FUNCTION_BLOCK AR_CLIENT_1_0 (* Send a REAL from an AR adapter as a remote OPC-UA write via CLIENT_1_0, buffered with a D_FF *)
  (* Standard: 61499-2; Description: Copyright (c) 2026 HR Agrartechnik GmbH This program and the accompanying materials are made available under the terms of the Eclipse Public License 2.0 which is available at https://www.eclipse.org/legal/epl-2.0/ SPDX-License-Identifier: EPL-2.0 *)
  (* Version 1.0, 2026-09-16, Franz Höpfinger, HR Agrartechnik GmbH, initial API and implementation and/or initial documentation - analog zu AX_CLIENT_1_0, REAL statt BOOL (fehlender Client-FB fuer Remote-Write eines REAL-Wertes, siehe BERICHT_2026-09-16_STG3_I1_I3_I4_I6_STALE_REMOTE_SUBSCRIBE.md Abschnitt 11). *)
  PACKAGE adapter::net;
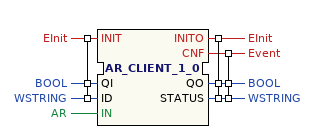
  EVENT_INPUT
    INIT : EInit WITH QI, ID; (* Initialization *)
  END_EVENT
  EVENT_OUTPUT
    INITO : EInit WITH QO, STATUS; (* Initialization Confirm *)
    CNF WITH QO, STATUS; (* Data was sent *)
  END_EVENT
  VAR_INPUT
    QI : BOOL;
    ID : WSTRING;
  END_VAR
  VAR_OUTPUT
    QO : BOOL;
    STATUS : WSTRING;
  END_VAR
  SOCKETS
    IN : adapter::types::unidirectional::AR; (* REAL to send *)
  END_SOCKETS
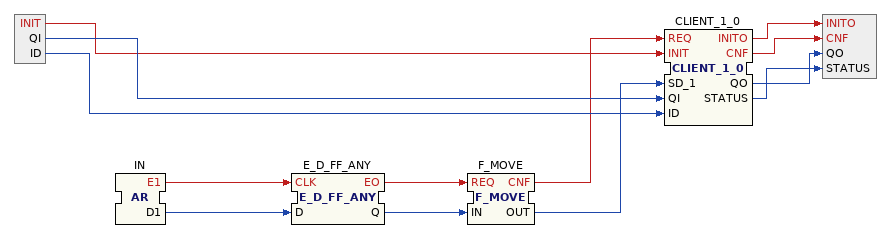
  FBS
    E_D_FF_ANY : iec61499::events::E_D_FF_ANY;
    F_MOVE : iec61131::selection::F_MOVE; {SET_ATTRIBUTE(DataType, REAL)}
    CLIENT_1_0 : iec61499::net::CLIENT_1_0;
  END_FBS
  EVENT_CONNECTIONS
    CLIENT_1_0.INITO TO INITO;
    CLIENT_1_0.CNF TO CNF;
    IN.E1 TO E_D_FF_ANY.CLK;
    E_D_FF_ANY.EO TO F_MOVE.REQ;
    F_MOVE.CNF TO CLIENT_1_0.REQ;
    INIT TO CLIENT_1_0.INIT;
  END_CONNECTIONS
  DATA_CONNECTIONS
    CLIENT_1_0.QO TO QO;
    CLIENT_1_0.STATUS TO STATUS;
    IN.D1 TO E_D_FF_ANY.D;
    E_D_FF_ANY.Q TO F_MOVE.IN;
    F_MOVE.OUT TO CLIENT_1_0.SD_1;
    QI TO CLIENT_1_0.QI;
    ID TO CLIENT_1_0.ID;
  END_CONNECTIONS
END_FUNCTION_BLOCK
